PROGRAM S_UnLoadWafer
VAR_INPUT
	bInit				:BOOL:=FALSE;// 初始化状态 busy/done/errDone
	bTrig				:BOOL:=FALSE;// 执行触发 信号
	bReset				:BOOL:=FALSE;// 报错 复位
	bPause				:BOOL:=FALSE;// 暂停 运行
	bStop				:BOOL:=FALSE;// 停止 运行
	bAbort				:BOOL:=FALSE;// 中止 运行
	
END_VAR
VAR_OUTPUT
	busy				:BOOL;
	done				:BOOL;
	errDone				:BOOL;
END_VAR
VAR
	actStep				:ActStepBase;
END_VAR
VAR
	i: INT;
	t1:ton;
	t2:ton;
	t3:ton;
	notchoose:BOOL;
	timeOutTime:TIME:= T#120S;
	ventTime:TIME:=T#25S;
	ventTimes:INT;
END_VAR

busy:=actStep.isBusy();
done:=actStep.isDone();
errDone:=actStep.isError();
actStep.Act_Pause(pause:=bPause);

IF bTrig THEN
	bTrig:=FALSE;
	IF NOT busy THEN
		actStep.Act_ex();
	END_IF
END_IF

//状态复位
IF bInit THEN
	bInit:=FALSE;
	Act_init_status();
END_IF

IF bAbort OR bStop THEN
	bAbort:=FALSE;
	bStop:=FALSE;
	Act_init_status();
	actStep.toZeroStep();
	gShowLogTextTitle:='NON';
END_IF
ActionRun(tempActStep:=actStep);

(*
---Trigger action
*)
METHOD Act_Ex : BOOL
VAR_INPUT
END_VAR
IF NOT busy THEN
	actStep.Act_ex();
	Act_Ex:=TRUE;
ELSE
	Act_Ex:=FALSE;
END_IF
END_METHOD

(*
---功能: 状态复位 busy/done/errDone;
*)
METHOD Act_Init_Status
VAR_INPUT
END_VAR
actStep.Act_Init();
END_METHOD

METHOD PRIVATE ActionRun
VAR_INPUT
	tempActStep:ITFActStep;
END_VAR
VAR_STAT//此处定义静态变量, 保证每次进入该函数时能够在线监控当前值
	tempStep:DINT;
END_VAR
tempStep:=tempActStep.getStep();
CASE tempStep OF
0:
	IF tempActStep.isEx() THEN
		tempActStep.setBusyFlag();
		tempActStep.toBeginStep();
	END_IF
	t1(IN:= FALSE );
	t2(IN:= FALSE );
	t3(IN:= FALSE );
10:
	gShowLogTextTitle:='UnLoad Wafer';
	IF gRunningState<>RunningStatus.eErrorState THEN
		tempActStep.addStep(10,FALSE);
	ELSE
		error_Trigger(105);
		IF gCtrlMode=ControlMode.eManualCtrMode THEN
			tempActStep.toErrDoneStep();
		END_IF
	END_IF
20:
	IF ControlMode.eManualCtrMode=gCtrlMode THEN
		tempActStep.addStep(40,FALSE);
	ELSIF( ControlMode.eAutoCtrMode=gCtrlMode) THEN
		tempActStep.addStep(40,FALSE);
	ELSE
		tempActStep.toErrDoneStep();
	END_IF
30:
	tempActStep.addStep(10,FALSE);
40:
	tempActStep.addStep(10,TRUE);
50:
	tempActStep.addStep(10,FALSE);
60:
	S_RoughPumping.Act_Init_Status();
	S_RoughPumping.Act_Ex();
	tempActStep.addStep(10,FALSE);
70:
	IF S_RoughPumping.done THEN
		gShowLogTextTitle:='UnLoad Wafer';
		tempActStep.addStep(10,FALSE);
	END_IF
	IF S_RoughPumping.errDone THEN
		tempActStep.toErrDoneStep();
	END_IF
80:
	tempActStep.addStep(20,TRUE);
100:
	IF gWaferMemoryState=1 OR gWaferMemoryState=2 THEN// 腔体有晶圆
		IF NOT gICP.I_WaferCheck THEN
			tempActStep.addStep(10,FALSE);
		ELSE
			error_Trigger(115);
			tempActStep.toErrDoneStep();
		END_IF
	ELSE
		gRunningLog.append(CONCAT('UnLoad Wafer POU Step:',DINT_TO_STRING(tempStep)));
		gRunningLog.append('UnLoad Wafer POU Run:Wafer In Chamber To Vent LoadLock');
		tempActStep.toStep(500,FALSE);// LoadLock有料，则直接判断UnLoad完成（或者衔接无料Vent的过程）
	END_IF
110:
	tempActStep.addStep(5,TRUE);
115:
	IF gICP.GateDoorValve.Act_Retract() AND gICP.VentValve.Act_Retract() THEN
		gRunningLog.append(CONCAT('UnLoad Wafer POU Step:',DINT_TO_STRING(tempStep)));
		gRunningLog.append('UnLoad Wafer POU Run:Gate Door Close And Vent Close');
		tempActStep.addStep(5,FALSE);
	END_IF
120:
	IF gICP.GateDoorValve.Get_Done_Ret() AND gICP.GateDoorRetSensor AND
       gICP.VentValve.Get_Done_Ret() AND NOT gICP.VentExtRelay THEN
	   gRunningLog.append(CONCAT('UnLoad Wafer POU Step:',DINT_TO_STRING(tempStep)));
	   gRunningLog.append('UnLoad Wafer POU Run:Gate Door Close Done And Vent Valve Close Done');
		tempActStep.addStep(10,FALSE);
	END_IF
130:
	IF gICP.ElectrodeCyl.Act_Retract() THEN
		gRunningLog.append(CONCAT('UnLoad Wafer POU Step:',DINT_TO_STRING(tempStep)));
		gRunningLog.append('UnLoad Wafer POU Run:ElectrodeCyl Dowm');
		tempActStep.addStep(10,FALSE);
	END_IF
140:
	IF gICP.ElectrodeCyl.Get_Done_Ret() AND gICP.ElectrodeCylRetSensor THEN
		gRunningLog.append(CONCAT('UnLoad Wafer POU Step:',DINT_TO_STRING(tempStep)));
		gRunningLog.append('UnLoad Wafer POU Run:ElectrodeCyl Dowm Done');
		tempActStep.addStep(10,FALSE);
	END_IF
150:
	tempActStep.addStep(10,FALSE);
160:
	tempActStep.addStep(10,TRUE);
170:
	IF gICP.LiftPinCyl.Act_Extend() THEN
		gRunningLog.append(CONCAT('UnLoad Wafer POU Step:',DINT_TO_STRING(tempStep)));
		gRunningLog.append('UnLoad Wafer POU Run:LiftPinCyl UP');
		tempActStep.addStep(10,FALSE);
	END_IF
180:
	IF gICP.LiftPinCyl.Get_Done_Ext() AND gICP.LiftPinExtSensor THEN
		gRunningLog.append(CONCAT('UnLoad Wafer POU Step:',DINT_TO_STRING(tempStep)));
		gRunningLog.append('UnLoad Wafer POU Run:LiftPinCyl UP Down');
		tempActStep.addStep(10,FALSE);
	END_IF
190:
	t1(IN:=TRUE,PT:=T#1S);
	IF t1.Q THEN
		t1(IN:= FALSE );
		t2(IN:= FALSE );
		t3(IN:= FALSE );
		tempActStep.addStep(10,FALSE);
	END_IF
200:
	tempActStep.addStep(10,FALSE);
210:
	tempActStep.addStep(10,TRUE);
220:
	IF NOT gICP.VentExtRelay AND gICP.ForlinLineValveExtRelay AND NOT gICP.RoughValveExtRelay THEN
		tempActStep.addStep(10,FALSE);
	ELSE
		error_Trigger(105);
		tempActStep.toStep(210,FALSE);
	END_IF
230://////////////准备破LoadLock
	IF gICP.LoadLockGauge.outputValue<gRoughtPumVaccum THEN // LL 真空满足
		IF NOT gICP.LoadLockGauge.error AND gICP.PDV.Act_Retract()  THEN
			tempActStep.toStep(340,FALSE);
			gRunningLog.append(CONCAT('UnLoad Wafer POU Step:',DINT_TO_STRING(tempStep)));
			gRunningLog.append(CONCAT('UnLoad Wafer POU Run:LL Pressure Arrive ',REAL_TO_STRING(gICP.LoadLockGauge.outputValue)));
		ELSE
			error_Trigger(105);
			tempActStep.toStep(210,FALSE);
		END_IF
	ELSE
		tempActStep.addStep(10,FALSE);
	END_IF
240:
	tempActStep.addStep(2,TRUE);
242:
	IF gICP.ForlinLineValve.Act_Retract() AND gICP.PDV.Act_Retract() THEN
		tempActStep.addStep(2,FALSE);
	END_IF
244:
	IF gICP.ForlinLineValve.Get_Done_Ret() AND (gICP.PDVCloseSensor OR gICP.PDV.Get_Done_Ret()) THEN
		tempActStep.addStep(2,FALSE);
	END_IF
246:
	tempActStep.addStep(4,TRUE);
250:
	IF gICP.SlowPummingValve.Act_Extend() AND gICP.FastPummingValve.Act_Retract() THEN
		gRunningLog.append(CONCAT('UnLoad Wafer POU Step:',DINT_TO_STRING(tempStep)));
		gRunningLog.append('UnLoad Wafer POU Run:SlowPummingValve Open and FastPummingValve Close');
		tempActStep.addStep(10,FALSE);
	END_IF
260:
	IF gICP.SlowPummingValve.Get_Done_Ext() AND gICP.FastPummingValve.Get_Done_Ret() THEN
		gRunningLog.append(CONCAT('UnLoad Wafer POU Step:',DINT_TO_STRING(tempStep)));
		gRunningLog.append('UnLoad Wafer POU Run:SlowPummingValve Open Done and FastPummingValve Close Done');
		tempActStep.addStep(10,FALSE);
	END_IF
270:
	t2(IN:=gICP.LoadLockGauge.outputValue<gLoadLockPumSVaccum,PT:=T#2S);
	IF t2.Q THEN
		t1(IN:= FALSE );
		t2(IN:= FALSE );
		t3(IN:= FALSE );
		gRunningLog.append(CONCAT('UnLoad Wafer POU Step:',DINT_TO_STRING(tempStep)));
		gRunningLog.append(CONCAT('UnLoad Wafer POU Run:LL Pressure Arrive ',REAL_TO_STRING(gICP.LoadLockGauge.outputValue)));
		tempActStep.addStep(10,FALSE);
	END_IF
280:
	IF gICP.SlowPummingValve.Act_Retract() AND gICP.FastPummingValve.Act_Extend() THEN
		gRunningLog.append(CONCAT('UnLoad Wafer POU Step:',DINT_TO_STRING(tempStep)));
		gRunningLog.append('UnLoad Wafer POU Run:SlowPummingValve Close and FastPummingValve Open');
		tempActStep.addStep(10,FALSE);
	END_IF
290:
	IF gICP.SlowPummingValve.Get_Done_Ret() AND gICP.FastPummingValve.Get_Done_Ext() THEN
		gRunningLog.append(CONCAT('UnLoad Wafer POU Step:',DINT_TO_STRING(tempStep)));
		gRunningLog.append('UnLoad Wafer POU Run:SlowPummingValve Close Done and FastPummingValve Open Done');
		tempActStep.addStep(10,FALSE);
	END_IF
300:
	t2(IN:=gICP.LoadLockGauge.outputValue<gRoughtPumVaccum,PT:=T#2S);
	IF t2.Q THEN
		t1(IN:= FALSE );
		t2(IN:= FALSE );
		t3(IN:= FALSE );
		gRunningLog.append(CONCAT('UnLoad Wafer POU Step:',DINT_TO_STRING(tempStep)));
		gRunningLog.append(CONCAT('UnLoad Wafer POU Run:LL Pressure Arrive ',REAL_TO_STRING(gICP.LoadLockGauge.outputValue)));
		tempActStep.addStep(10,FALSE);
	END_IF
310:
	tempActStep.addStep(10,TRUE);
320:
	IF gICP.SlowPummingValve.Act_Retract() AND gICP.FastPummingValve.Act_Retract() AND gICP.PDV.Act_Retract() THEN
		gRunningLog.append(CONCAT('UnLoad Wafer POU Step:',DINT_TO_STRING(tempStep)));
		gRunningLog.append('UnLoad Wafer POU Run:SlowPummingValve Close | FastPummingValve Close | PDV Open');
		tempActStep.addStep(10,FALSE);
	END_IF
330:
	IF gICP.SlowPummingValve.Get_Done_Ret() AND gICP.FastPummingValve.Get_Done_Ret() AND (gICP.PDV.Get_Done_Ret() OR gICP.PDVCloseSensor) THEN
		gRunningLog.append(CONCAT('UnLoad Wafer POU Step:',DINT_TO_STRING(tempStep)));
		gRunningLog.append('UnLoad Wafer POU Run:SlowPummingValve Close Done | FastPummingValve Close Done | PDV Open Done');
		tempActStep.addStep(10,FALSE);
	END_IF
340:
	IF (gICP.PDV.Get_Done_Ret() OR gICP.PDVCloseSensor) THEN
		tempActStep.addStep(10,TRUE);
	END_IF
350:
	IF gICP.GateDoorValve.Act_Extend() THEN
		gRunningLog.append(CONCAT('UnLoad Wafer POU Step:',DINT_TO_STRING(tempStep)));
		gRunningLog.append('UnLoad Wafer POU Run:Gate Door Open');
		tempActStep.addStep(5,FALSE);
	END_IF
355:
	IF gICP.GateDoorValve.Get_Done_Ext() AND gICP.GateDoorExtSensor THEN
		gRunningLog.append(CONCAT('UnLoad Wafer POU Step:',DINT_TO_STRING(tempStep)));
		gRunningLog.append('UnLoad Wafer POU Run:Gate Door Open Done');
		tempActStep.addStep(5,FALSE);
	END_IF
360:
	IF gICP.HeMFC_ActFlow<1 AND gICP.HeCheckGaugeReal<1 AND NOT gICP.HeINExtRelay AND NOT gICP.HePumExtRelay THEN
		tempActStep.addStep(1,FALSE);
	ELSE
		tempActStep.addStep(10,FALSE);
	END_IF
361:
	tempActStep.addStep(1,TRUE);
362:
	IF gICP.HeINValve.Act_Retract() THEN
		tempActStep.addStep(1,FALSE);
	END_IF
363:
	IF gICP.HeINValve.Get_Done_Ret() THEN
		tempActStep.addStep(1,FALSE);
	END_IF
364:
	tempActStep.addStep(1,TRUE);
365:
	IF gICP.HePumValve.Act_Extend() THEN
		tempActStep.addStep(1,FALSE);
	END_IF
366:
	IF gICP.HePumValve.Get_Done_Ext() THEN
		tempActStep.addStep(1,FALSE);
	END_IF
367:
	t2(IN:=TRUE ,PT:=T#2S);
	IF t2.Q THEN
		t1(IN:= FALSE );
		t2(IN:= FALSE );
		t3(IN:= FALSE );
		tempActStep.addStep(1,FALSE);
	END_IF
368:
	t1(IN:=gICP.HeMFC_ActFlow<1 AND gICP.HeCheckGaugeReal<1 ,PT:=T#2S);
	IF t1.Q THEN
		t1(IN:= FALSE );
		t2(IN:= FALSE );
		t3(IN:= FALSE );
		gICP.HePumValve.Act_Retract();
		tempActStep.addStep(2,FALSE);
	END_IF
370:
	IF gICP.ElectrodeCyl.Act_Retract() AND gICP.HePumValve.Get_Done_Ret() THEN
		gRunningLog.append(CONCAT('UnLoad Wafer POU Step:',DINT_TO_STRING(tempStep)));
		gRunningLog.append('UnLoad Wafer POU Run:ElectrodeCyl Down');
		tempActStep.addStep(2,FALSE);
	END_IF
372:
	IF gICP.ElectrodeCyl.Get_Done_Ret() THEN
		gRunningLog.append(CONCAT('UnLoad Wafer POU Step:',DINT_TO_STRING(tempStep)));
		gRunningLog.append('UnLoad Wafer POU Run:ElectrodeCyl Down Done');
		tempActStep.addStep(2,FALSE);
	END_IF
374:
	tempActStep.addStep(2,TRUE);
376:
	IF gICP.LiftPinCyl.Act_Extend() THEN
		gRunningLog.append(CONCAT('UnLoad Wafer POU Step:',DINT_TO_STRING(tempStep)));
		gRunningLog.append('UnLoad Wafer POU Run:LiftPinCyl UP');
		tempActStep.addStep(2,FALSE);
	END_IF
378:
	IF gICP.LiftPinCyl.Get_Done_Ext() THEN
		gRunningLog.append(CONCAT('UnLoad Wafer POU Step:',DINT_TO_STRING(tempStep)));
		gRunningLog.append('UnLoad Wafer POU Run:LiftPinCyl UP Done');
		tempActStep.addStep(1,FALSE);
	END_IF
379:
	tempActStep.addStep(1,TRUE);
380:
	tempActStep.addStep(20,FALSE);
400:
	IF gICP.ARM.Act_IN_Auto() THEN
		gRunningLog.append(CONCAT('UnLoad Wafer POU Step:',DINT_TO_STRING(tempStep)));
		gRunningLog.append('UnLoad Wafer POU Run:ARM IN');
		tempActStep.addStep(10,FALSE);
	END_IF
410:
	IF NOT gICP.I_ARMHome THEN// 手臂当前不应该在原点位置
		tempActStep.addStep(10,FALSE);
	END_IF
420:
	t1(IN:=gICP.ARM.Get_Done_IN() AND NOT gICP.ARM.busy AND ABS(gICP.ARM.actpos-gARMPosition)<=1 ,PT:=T#2S);
	IF t1.Q THEN
		t1(IN:= FALSE );
		t2(IN:= FALSE );
		t3(IN:= FALSE );
		gRunningLog.append(CONCAT('UnLoad Wafer POU Step:',DINT_TO_STRING(tempStep)));
		gRunningLog.append('UnLoad Wafer POU Run:ARM IN Done');
		tempActStep.addStep(10,FALSE);
		RETURN;
	END_IF
	t2(IN:=TRUE,PT:=T#20S);
	IF t2.Q THEN
		t1(IN:= FALSE );
		t2(IN:= FALSE );
		t3(IN:= FALSE );
		error_Trigger(114);
		tempActStep.toStep(379,FALSE);
		RETURN;
	END_IF
430:
	tempActStep.addStep(10,TRUE);
440:
	IF gICP.LiftPinCyl.Act_Retract() THEN
		gRunningLog.append(CONCAT('UnLoad Wafer POU Step:',DINT_TO_STRING(tempStep)));
		gRunningLog.append('UnLoad Wafer POU Run:LiftPinCyl Down');
		tempActStep.addStep(10,FALSE);
	END_IF
450:
	IF gICP.LiftPinCyl.Get_Done_Ret() AND gICP.LiftPinRetSensor THEN
		gRunningLog.append(CONCAT('UnLoad Wafer POU Step:',DINT_TO_STRING(tempStep)));
		gRunningLog.append('UnLoad Wafer POU Run:LiftPinCyl Down Done');
		// 记忆状态更新
		gWaferMemoryState:=0;
		ups_CX51X0.Act_Wrtie();
		tempActStep.addStep(10,FALSE);
	END_IF
460:
	tempActStep.addStep(10,TRUE);
470:
	IF gICP.ARM.Act_HOME_Auto() THEN
		gRunningLog.append(CONCAT('UnLoad Wafer POU Step:',DINT_TO_STRING(tempStep)));
		gRunningLog.append('UnLoad Wafer POU Run:ARM Home');
		tempActStep.addStep(10,FALSE);
	END_IF
480:
	IF gICP.ARM.Get_Done_HOME() AND gICP.I_ARMHome AND ABS(gICP.ARM.actpos-0)<=1 AND NOT gICP.ARM.busy THEN// 手臂当前不应该在原点位置
		gRunningLog.append(CONCAT('UnLoad Wafer POU Step:',DINT_TO_STRING(tempStep)));
		gRunningLog.append('UnLoad Wafer POU Run:ARM Home Done');
		tempActStep.addStep(10,FALSE);
	END_IF
490:
	t2(IN:=TRUE,PT:=T#2S);
	IF t2.Q THEN
		t1(IN:= FALSE );
		t2(IN:= FALSE );
		t3(IN:= FALSE );
		tempActStep.addStep(10,FALSE);
		RETURN;
	END_IF
500:
	ventTimes:=1;
	tempActStep.addStep(10,TRUE);
510:
	IF gICP.GateDoorValve.Act_Retract() THEN
		gRunningLog.append(CONCAT('UnLoad Wafer POU Step:',DINT_TO_STRING(tempStep)));
		gRunningLog.append('UnLoad Wafer POU Run:GateDoorValve Close');
		tempActStep.addStep(10,FALSE);
	END_IF
520:
	IF gICP.GateDoorValve.Get_Done_Ret() AND gICP.GateDoorRetSensor THEN
		gRunningLog.append(CONCAT('UnLoad Wafer POU Step:',DINT_TO_STRING(tempStep)));
		gRunningLog.append('UnLoad Wafer POU Run:GateDoorValve Close Done');
		tempActStep.addStep(10,FALSE);
	END_IF
530:
	tempActStep.addStep(10,TRUE);
540:
	IF  gICP.GateDoorValve.Act_Retract() AND 
	    gICP.SlowPummingValve.Act_Retract() AND 
	    gICP.FastPummingValve.Act_Retract() THEN
		tempActStep.addStep(10,FALSE);
	END_IF
550:
	IF gICP.GateDoorValve.Get_Done_Ret() AND gICP.GateDoorRetSensor AND
	   gICP.SlowPummingValve.Get_Done_Ret() AND NOT gICP.SlowPummingExtRelay AND
	   gICP.FastPummingValve.Get_Done_Ret() AND NOT gICP.FastPummingExtRelay THEN
		tempActStep.addStep(10,FALSE);
	END_IF
560:
	IF gICP.VentValve.Act_Extend() THEN
		gRunningLog.append(CONCAT('UnLoad Wafer POU Step:',DINT_TO_STRING(tempStep)));
		gRunningLog.append('UnLoad Wafer POU Run:VentValve Open');
		tempActStep.addStep(10,FALSE);
	END_IF
570:
	IF gICP.VentValve.Get_Done_Ext() THEN
		gRunningLog.append(CONCAT('UnLoad Wafer POU Step:',DINT_TO_STRING(tempStep)));
		gRunningLog.append('UnLoad Wafer POU Run:VentValve Open Done');
		tempActStep.addStep(10,FALSE);
	END_IF
580:
	t2(IN:=gICP.LoadLockGauge.outputValue>gATMPressure,PT:=ventTime/ventTimes);
	IF t2.Q OR NOT gICP.I_LLSwitch THEN
		t1(IN:= FALSE );
		t2(IN:= FALSE );
		t3(IN:= FALSE );
		gRunningLog.append(CONCAT('UnLoad Wafer POU Step:',DINT_TO_STRING(tempStep)));
		gRunningLog.append(CONCAT('UnLoad Wafer POU Run:LL Pressure Arrive ',REAL_TO_STRING(gICP.LoadLockGauge.outputValue)));
		tempActStep.addStep(10,FALSE);
	END_IF
590:
	tempActStep.addStep(10,TRUE);
600:
	IF gICP.VentValve.Act_Retract() THEN
		gRunningLog.append(CONCAT('UnLoad Wafer POU Step:',DINT_TO_STRING(tempStep)));
		gRunningLog.append('UnLoad Wafer POU Run:VentValve Close');
		tempActStep.addStep(10,FALSE);
	END_IF
610:
	IF gICP.VentValve.Get_Done_Ret() THEN
		gRunningLog.append(CONCAT('UnLoad Wafer POU Step:',DINT_TO_STRING(tempStep)));
		gRunningLog.append('UnLoad Wafer POU Run:VentValve Close Done');
		tempActStep.addStep(10,FALSE);
	END_IF
620:
	t1(IN:=TRUE,PT:=T#1S);
	IF t1.Q THEN
		t1(IN:= FALSE );
		t2(IN:= FALSE );
		t3(IN:= FALSE );
		gRunningLog.append('UnLoad Wafer POU Run:Wait for the wafer to be removed');
		tempActStep.addStep(10,FALSE);
	END_IF
630:
	t2(IN:=NOT gICP.I_WaferCheck AND gICP.I_LLSwitch,PT:=T#1S);// 拿走晶圆，且关上盖子
	IF t2.Q THEN
		t1(IN:= FALSE );
		t2(IN:= FALSE );
		t3(IN:= FALSE );
		gRunningLog.append(CONCAT('UnLoad Wafer POU Step:',DINT_TO_STRING(tempStep)));
		gRunningLog.append('UnLoad Wafer POU Run:Wafer tack out and close LL');
		tempActStep.addStep(10,FALSE);
		RETURN;
	END_IF
	t3(IN:=TRUE,PT:=timeOutTime);
	IF t3.Q THEN
		error_Trigger(114);
		ventTimes:=3;
		tempActStep.toStep(530,FALSE);
	END_IF
640:
	IF gICP.ForlinLineValve.Act_Extend() THEN
		gRunningLog.append(CONCAT('UnLoad Wafer POU Step:',DINT_TO_STRING(tempStep)));
		gRunningLog.append('UnLoad Wafer POU Run:ForLineValve Open');
		tempActStep.addStep(10,FALSE);
	END_IF
650:
	IF gICP.ForlinLineValve.Get_Done_Ext() THEN
		gRunningLog.append(CONCAT('UnLoad Wafer POU Step:',DINT_TO_STRING(tempStep)));
		gRunningLog.append('UnLoad Wafer POU Run:ForLineValve Open Done');
		tempActStep.addStep(10,FALSE);
	END_IF
660:
	tempActStep.addStep(10,TRUE);
670:
	IF gICP.PDV.Act_Open() THEN
		gRunningLog.append(CONCAT('UnLoad Wafer POU Step:',DINT_TO_STRING(tempStep)));
		gRunningLog.append('UnLoad Wafer POU Run:PDV Open');
		tempActStep.addStep(10,FALSE);
	END_IF
680:
	IF gICP.PDV.Get_Done_Ext() OR gICP.PDVOpenSensor THEN
		gRunningLog.append(CONCAT('UnLoad Wafer POU Step:',DINT_TO_STRING(tempStep)));
		gRunningLog.append('UnLoad Wafer POU Run:PDV Open Done');
		tempActStep.addStep(10,FALSE);
	END_IF
690:
	// 记忆状态更新
	gWaferMemoryState:=0;
	ups_CX51X0.Act_Wrtie();
	gRunningLog.append(CONCAT('UnLoad Wafer POU Step:',DINT_TO_STRING(tempStep)));
	gRunningLog.append('UnLoad Wafer POU Run:----Finish----');
	tempActStep.toDoneStep();
1000:
	tempActStep.toDoneStep();

60000://Done
	tempActStep.setDoneFlag();
	tempActStep.toZeroStep();
	
65000://Error
	tempActStep.setErrDoneFlag();
	tempActStep.toZeroStep();
	IF gICP.VentExtRelay THEN
		gICP.VentValve.Act_Retract();
	END_IF
END_CASE
END_METHOD

END_PROGRAM

(* stored: Version 1.1.0.1, ProductVersion 3.1.4024.12
   POU S_UnLoadWafer: Id {fa77902a-dbc1-441b-b684-82dc0496a7e0}, SpecialFunc None
   Folder Private: Id {17a15fc6-a961-4d42-a3a3-e318d1c15368}
   Method Act_Ex: Id {a5e6d000-ba96-49d1-bed6-3e5af4359ca2}
   Method Act_Init_Status: Id {ce65aa57-518f-4da3-8a89-78a9dfe8310a}
   Method ActionRun: Id {46efe462-2ef3-4af6-8cee-fd21614ff578} *)
